(* Logix 5000 project; controller DispersionPlc vendor 1 type 14 code 108 rev 34.11; software revision 34.01; part 15 of 22 *)
(* tags used below, declared in another part *)
   _JISdebug : DINT;
   _Placeholder : DINT;
   AFI : BOOL;
   Estop_Disp : ALIAS FOR Local:3:I.Data.1;
   FQIC_4302_11_CurrentTrasferredLb : DINT;
   FQIC_4302_11_Reset : BOOL;
   FQIC_4302_11_TransferSetpoint : DINT;
   FQIC_4302_11_TransferStopValueLb : DINT;
   GenPurp : AStd_GeneralPurp;
   HS_S51_1 : AStd_DiscreteInput;
   HS_S51_1_AOI : AStd_DI_AOI;
   HS_S51_1_IRaw : BOOL;
   HS_S51_2 : AStd_DiscreteInput;
   HS_S51_2_AOI : AStd_DI_AOI;
   LAH_4302_11 : BOOL;   // Truck Loading Level Alarm High Probe
   LS_S51_1 : AStd_DiscreteInput;
   LS_S51_1_AOI : AStd_DI_AOI;
   LS_S51_1_IRaw : BOOL;
   LVL_W2_High : ALIAS FOR Local:1:I.Data[1].22;
   LVL_W4_High : ALIAS FOR Local:1:I.Data[1].23;
   PackTransferCompletePB : BOOL;
   RG_T51 : REAL;
   S4352_Phase_Circulation : AStd_PLI;
   S4352_Phase_Packaging_Transfer : AStd_PLI;
   S4352_Phase_Packaging_Transfer_AOI : AStd_PLI_AOI;
   S4352_Phase_TT_Transfer : AStd_PLI;
   S4352_Phase_TT_Transfer_AOI : AStd_PLI_AOI;
   S52TotalizerBypassPB : BOOL;
   SPARE_I_1_4_6 : ALIAS FOR Local:1:I.Data[4].6;
   SPARE_O_1_1_2 : ALIAS FOR Local:1:O.Data[1].2;
   SPARE_O_1_1_3 : ALIAS FOR Local:1:O.Data[1].3;
   SV_S52_2 : AStd_VlvOC;
   T4302_Phase_S52_Transfer : AStd_PLI;
   TIT_S51_1 : AStd_AnalogInput;
   TIT_S51_1_AOI : AStd_AI_AOI;
   TIT_S51_1_Raw : DINT;
   TIT_S51_2 : AStd_AnalogInput;
   TIT_S51_3 : AStd_AnalogInput;
   XV_4302_12 : AStd_VlvOC;
   XV_4302_13 : AStd_VlvOC;
   XV_S51_1 : AStd_VlvOC;
   XV_S51_1_AOI : AStd_VlvOC_AOI;
   XV_S51_1_IOpn : BOOL;
   XV_S51_1_OCls : BOOL;
   XV_S51_2 : AStd_VlvOC;
   XV_S51_2_AOI : AStd_VlvOC_AOI;
   XV_S51_2_ClsI : BOOL;
   XV_S51_2_IOpn : BOOL;
   XV_S51_2_OCls : BOOL;
   XV_S51_2CloseC : BOOL;
   XV_S51_2OpenC : BOOL;
   XV_S51_3 : AStd_VlvOC;
   XV_S51_3_AOI : AStd_VlvOC_AOI;
   XV_S51_3_IOpn : BOOL;
   XV_S51_3_OCls : BOOL;
   XV_S51_3CloseC : BOOL;
   XV_S51_3OpenC : BOOL;
   XV_S51_4 : AStd_VlvOC;
   XV_S51_4_AOI : AStd_VlvOC_AOI;
   XV_S51_4_IOpn : BOOL;
   XV_S51_4_OCls : BOOL;
   XV_S52_1 : AStd_VlvOC;
   XV_S52_2 : AStd_VlvOC;
(* Unit_S4352, continued *)

ROUTINE Phase_Packaging_Transfer   (* ladder *)
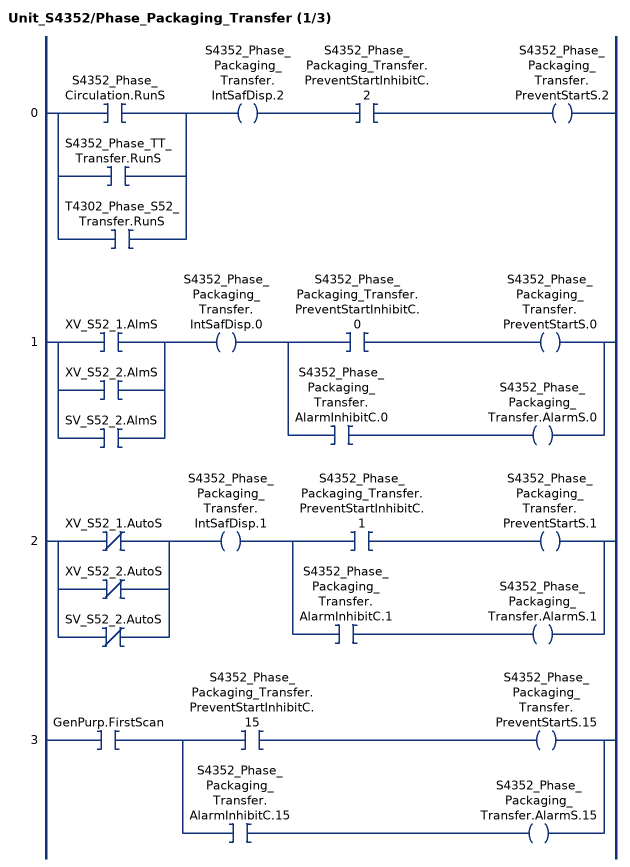
   0: [XIC(S4352_Phase_Circulation.RunS) ,XIC(S4352_Phase_TT_Transfer.RunS) ,XIC(T4302_Phase_S52_Transfer.RunS) ]OTE(S4352_Phase_Packaging_Transfer.IntSafDisp.2)XIC(S4352_Phase_Packaging_Transfer.PreventStartInhibitC.2)OTE(S4352_Phase_Packaging_Transfer.PreventStartS.2);
   1: [XIC(XV_S52_1.AlmS) ,XIC(XV_S52_2.AlmS) ,XIC(SV_S52_2.AlmS) ]OTE(S4352_Phase_Packaging_Transfer.IntSafDisp.0)[XIC(S4352_Phase_Packaging_Transfer.PreventStartInhibitC.0) OTE(S4352_Phase_Packaging_Transfer.PreventStartS.0) ,XIC(S4352_Phase_Packaging_Transfer.AlarmInhibitC.0) OTE(S4352_Phase_Packaging_Transfer.AlarmS.0) ];
   2: [XIO(XV_S52_1.AutoS) ,XIO(XV_S52_2.AutoS) ,XIO(SV_S52_2.AutoS) ]OTE(S4352_Phase_Packaging_Transfer.IntSafDisp.1)[XIC(S4352_Phase_Packaging_Transfer.PreventStartInhibitC.1) OTE(S4352_Phase_Packaging_Transfer.PreventStartS.1) ,XIC(S4352_Phase_Packaging_Transfer.AlarmInhibitC.1) OTE(S4352_Phase_Packaging_Transfer.AlarmS.1) ];
   3: XIC(GenPurp.FirstScan)[XIC(S4352_Phase_Packaging_Transfer.PreventStartInhibitC.15) OTE(S4352_Phase_Packaging_Transfer.PreventStartS.15) ,XIC(S4352_Phase_Packaging_Transfer.AlarmInhibitC.15) OTE(S4352_Phase_Packaging_Transfer.AlarmS.15) ];
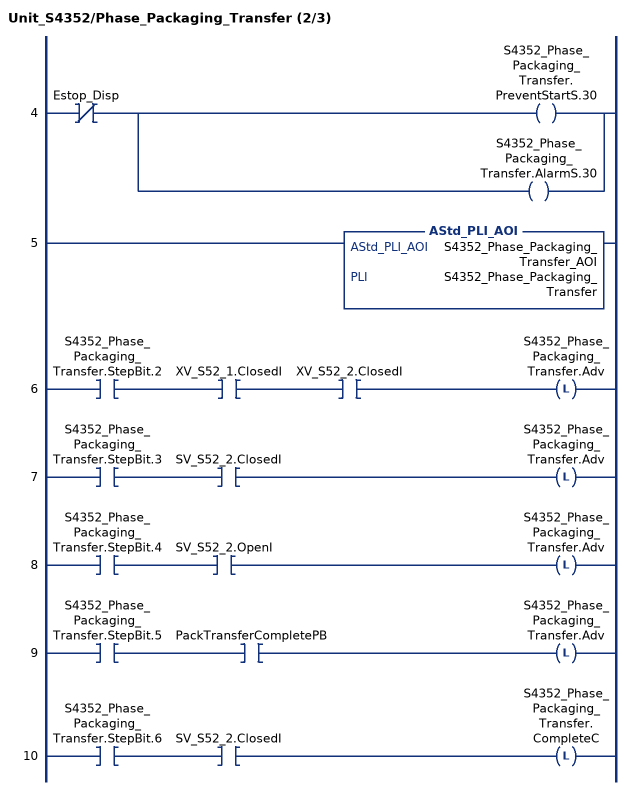
   4: XIO(Estop_Disp)[OTE(S4352_Phase_Packaging_Transfer.PreventStartS.30) ,OTE(S4352_Phase_Packaging_Transfer.AlarmS.30) ];
   5: AStd_PLI_AOI(S4352_Phase_Packaging_Transfer_AOI,S4352_Phase_Packaging_Transfer);
   6: XIC(S4352_Phase_Packaging_Transfer.StepBit.2)XIC(XV_S52_1.ClosedI)XIC(XV_S52_2.ClosedI)OTL(S4352_Phase_Packaging_Transfer.Adv);
   7: XIC(S4352_Phase_Packaging_Transfer.StepBit.3)XIC(SV_S52_2.ClosedI)OTL(S4352_Phase_Packaging_Transfer.Adv);
   8: XIC(S4352_Phase_Packaging_Transfer.StepBit.4)XIC(SV_S52_2.OpenI)OTL(S4352_Phase_Packaging_Transfer.Adv);
   9: XIC(S4352_Phase_Packaging_Transfer.StepBit.5)XIC(PackTransferCompletePB)OTL(S4352_Phase_Packaging_Transfer.Adv);
   10: XIC(S4352_Phase_Packaging_Transfer.StepBit.6)XIC(SV_S52_2.ClosedI)OTL(S4352_Phase_Packaging_Transfer.CompleteC);
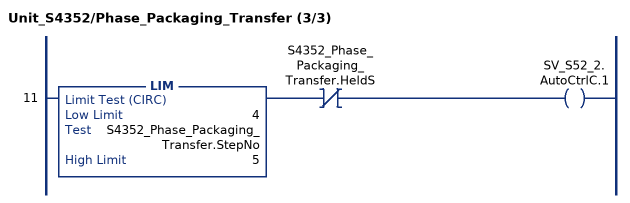
   11: LIM(4,S4352_Phase_Packaging_Transfer.StepNo,5)XIO(S4352_Phase_Packaging_Transfer.HeldS)OTE(SV_S52_2.AutoCtrlC.1);
END_ROUTINE

ROUTINE Phase_TT_Transfer   (* ladder *)
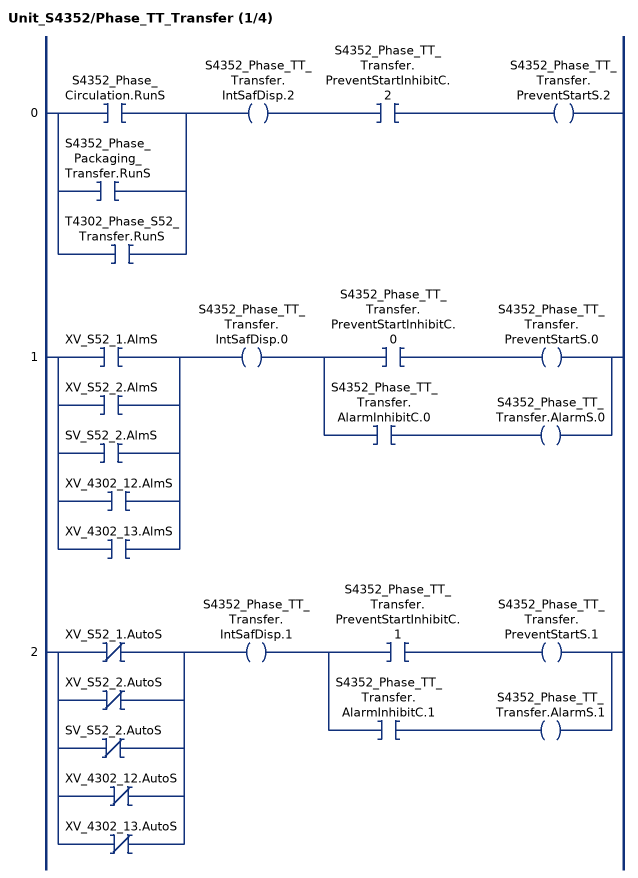
   0: [XIC(S4352_Phase_Circulation.RunS) ,XIC(S4352_Phase_Packaging_Transfer.RunS) ,XIC(T4302_Phase_S52_Transfer.RunS) ]OTE(S4352_Phase_TT_Transfer.IntSafDisp.2)XIC(S4352_Phase_TT_Transfer.PreventStartInhibitC.2)OTE(S4352_Phase_TT_Transfer.PreventStartS.2);
   1: [XIC(XV_S52_1.AlmS) ,XIC(XV_S52_2.AlmS) ,XIC(SV_S52_2.AlmS) ,XIC(XV_4302_12.AlmS) ,XIC(XV_4302_13.AlmS) ]OTE(S4352_Phase_TT_Transfer.IntSafDisp.0)[XIC(S4352_Phase_TT_Transfer.PreventStartInhibitC.0) OTE(S4352_Phase_TT_Transfer.PreventStartS.0) ,XIC(S4352_Phase_TT_Transfer.AlarmInhibitC.0) OTE(S4352_Phase_TT_Transfer.AlarmS.0) ];
   2: [XIO(XV_S52_1.AutoS) ,XIO(XV_S52_2.AutoS) ,XIO(SV_S52_2.AutoS) ,XIO(XV_4302_12.AutoS) ,XIO(XV_4302_13.AutoS) ]OTE(S4352_Phase_TT_Transfer.IntSafDisp.1)[XIC(S4352_Phase_TT_Transfer.PreventStartInhibitC.1) OTE(S4352_Phase_TT_Transfer.PreventStartS.1) ,XIC(S4352_Phase_TT_Transfer.AlarmInhibitC.1) OTE(S4352_Phase_TT_Transfer.AlarmS.1) ];
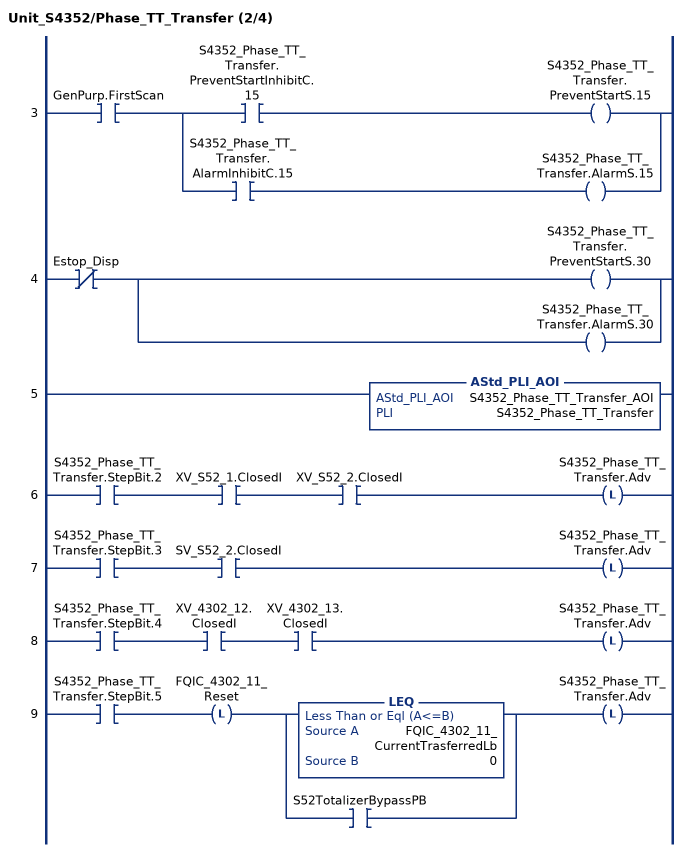
   3: XIC(GenPurp.FirstScan)[XIC(S4352_Phase_TT_Transfer.PreventStartInhibitC.15) OTE(S4352_Phase_TT_Transfer.PreventStartS.15) ,XIC(S4352_Phase_TT_Transfer.AlarmInhibitC.15) OTE(S4352_Phase_TT_Transfer.AlarmS.15) ];
   4: XIO(Estop_Disp)[OTE(S4352_Phase_TT_Transfer.PreventStartS.30) ,OTE(S4352_Phase_TT_Transfer.AlarmS.30) ];
   5: AStd_PLI_AOI(S4352_Phase_TT_Transfer_AOI,S4352_Phase_TT_Transfer);
   6: XIC(S4352_Phase_TT_Transfer.StepBit.2)XIC(XV_S52_1.ClosedI)XIC(XV_S52_2.ClosedI)OTL(S4352_Phase_TT_Transfer.Adv);
   7: XIC(S4352_Phase_TT_Transfer.StepBit.3)XIC(SV_S52_2.ClosedI)OTL(S4352_Phase_TT_Transfer.Adv);
   8: XIC(S4352_Phase_TT_Transfer.StepBit.4)XIC(XV_4302_12.ClosedI)XIC(XV_4302_13.ClosedI)OTL(S4352_Phase_TT_Transfer.Adv);
   9: XIC(S4352_Phase_TT_Transfer.StepBit.5)OTL(FQIC_4302_11_Reset)[LEQ(FQIC_4302_11_CurrentTrasferredLb,0) ,XIC(S52TotalizerBypassPB) ]OTL(S4352_Phase_TT_Transfer.Adv);
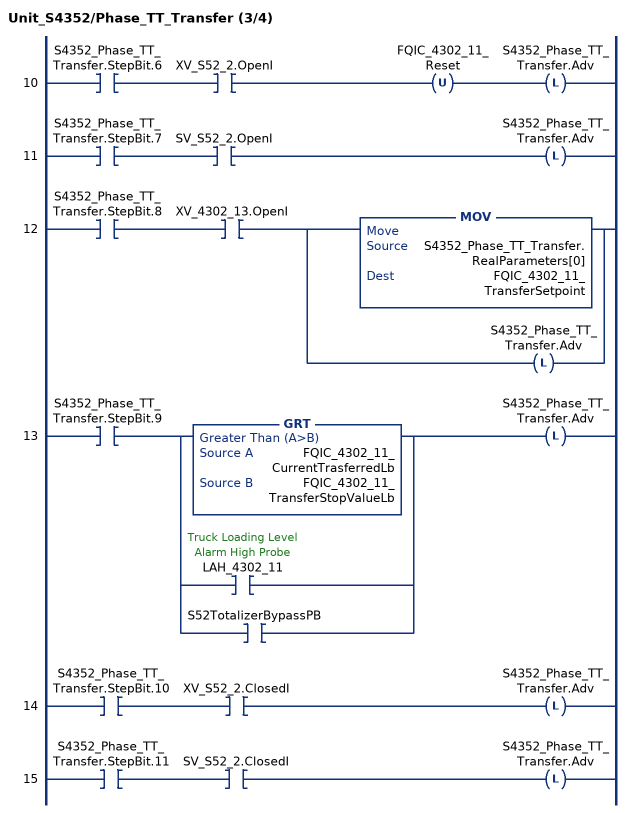
   10: XIC(S4352_Phase_TT_Transfer.StepBit.6)XIC(XV_S52_2.OpenI)OTU(FQIC_4302_11_Reset)OTL(S4352_Phase_TT_Transfer.Adv);
   11: XIC(S4352_Phase_TT_Transfer.StepBit.7)XIC(SV_S52_2.OpenI)OTL(S4352_Phase_TT_Transfer.Adv);
   12: XIC(S4352_Phase_TT_Transfer.StepBit.8)XIC(XV_4302_13.OpenI)[MOV(S4352_Phase_TT_Transfer.RealParameters[0],FQIC_4302_11_TransferSetpoint) ,OTL(S4352_Phase_TT_Transfer.Adv) ];
   13: XIC(S4352_Phase_TT_Transfer.StepBit.9)[GRT(FQIC_4302_11_CurrentTrasferredLb,FQIC_4302_11_TransferStopValueLb) ,XIC(LAH_4302_11) ,XIC(S52TotalizerBypassPB) ]OTL(S4352_Phase_TT_Transfer.Adv);
   14: XIC(S4352_Phase_TT_Transfer.StepBit.10)XIC(XV_S52_2.ClosedI)OTL(S4352_Phase_TT_Transfer.Adv);
   15: XIC(S4352_Phase_TT_Transfer.StepBit.11)XIC(SV_S52_2.ClosedI)OTL(S4352_Phase_TT_Transfer.Adv);
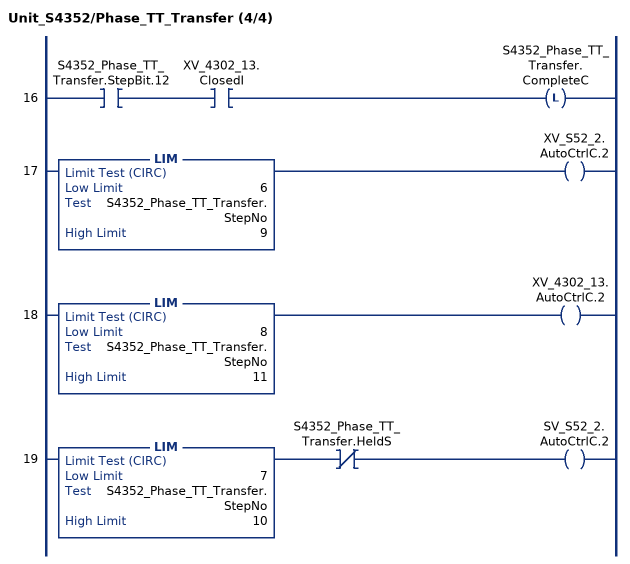
   16: XIC(S4352_Phase_TT_Transfer.StepBit.12)XIC(XV_4302_13.ClosedI)OTL(S4352_Phase_TT_Transfer.CompleteC);
   17: LIM(6,S4352_Phase_TT_Transfer.StepNo,9)OTE(XV_S52_2.AutoCtrlC.2);
   18: LIM(8,S4352_Phase_TT_Transfer.StepNo,11)OTE(XV_4302_13.AutoCtrlC.2);
   19: LIM(7,S4352_Phase_TT_Transfer.StepNo,10)XIO(S4352_Phase_TT_Transfer.HeldS)OTE(SV_S52_2.AutoCtrlC.2);
END_ROUTINE
END_PROGRAM

PROGRAM Unit_S51   (* main routine MainRoutine *)

ROUTINE Device_HS_S51_1   (* ladder *)
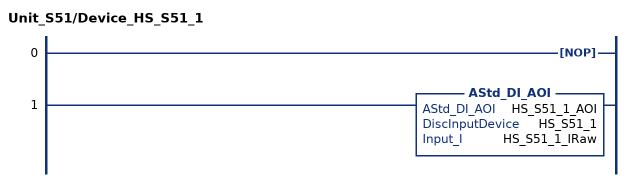
   0: NOP();
   1: AStd_DI_AOI(HS_S51_1_AOI,HS_S51_1,HS_S51_1_IRaw);
END_ROUTINE

ROUTINE Device_HS_S51_2   (* ladder *)
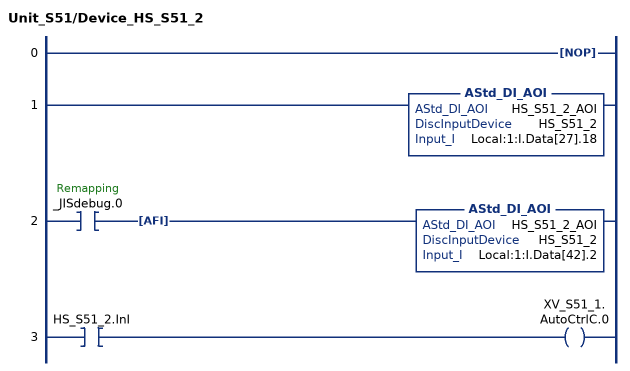
   0: NOP();
   1: AStd_DI_AOI(HS_S51_2_AOI,HS_S51_2,Local:1:I.Data[27].18);
   2: XIC(_JISdebug.0)AFI()AStd_DI_AOI(HS_S51_2_AOI,HS_S51_2,Local:1:I.Data[42].2);
   3: XIC(HS_S51_2.InI)OTE(XV_S51_1.AutoCtrlC.0);
END_ROUTINE

ROUTINE Device_LS_S51_1   (* ladder *)
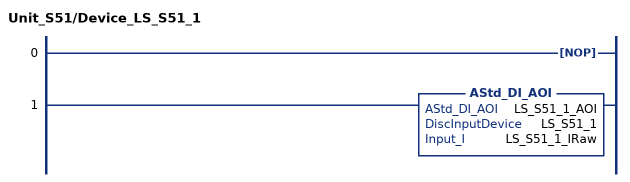
   0: NOP();
   1: AStd_DI_AOI(LS_S51_1_AOI,LS_S51_1,LS_S51_1_IRaw);
END_ROUTINE

ROUTINE Device_TIT_S51_1   (* ladder *)
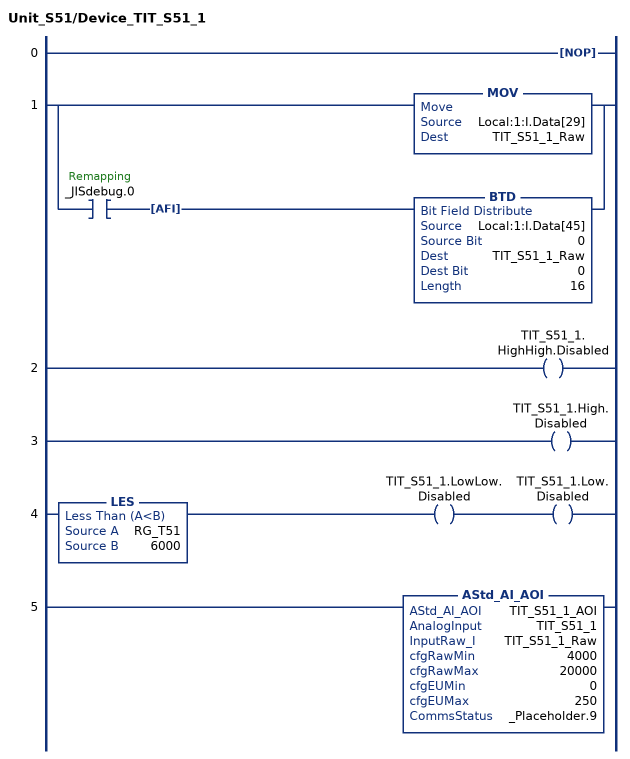
   0: NOP();
   1: [MOV(Local:1:I.Data[29],TIT_S51_1_Raw) ,XIC(_JISdebug.0) AFI() BTD(Local:1:I.Data[45],0,TIT_S51_1_Raw,0,16) ];
   2: OTE(TIT_S51_1.HighHigh.Disabled);
   3: OTE(TIT_S51_1.High.Disabled);
   4: LES(RG_T51,6000)OTE(TIT_S51_1.LowLow.Disabled)OTE(TIT_S51_1.Low.Disabled);
   5: AStd_AI_AOI(TIT_S51_1_AOI,TIT_S51_1,TIT_S51_1_Raw,4000,20000,0,250,_Placeholder.9);
END_ROUTINE

ROUTINE Device_XV_S51_1   (* ladder *)
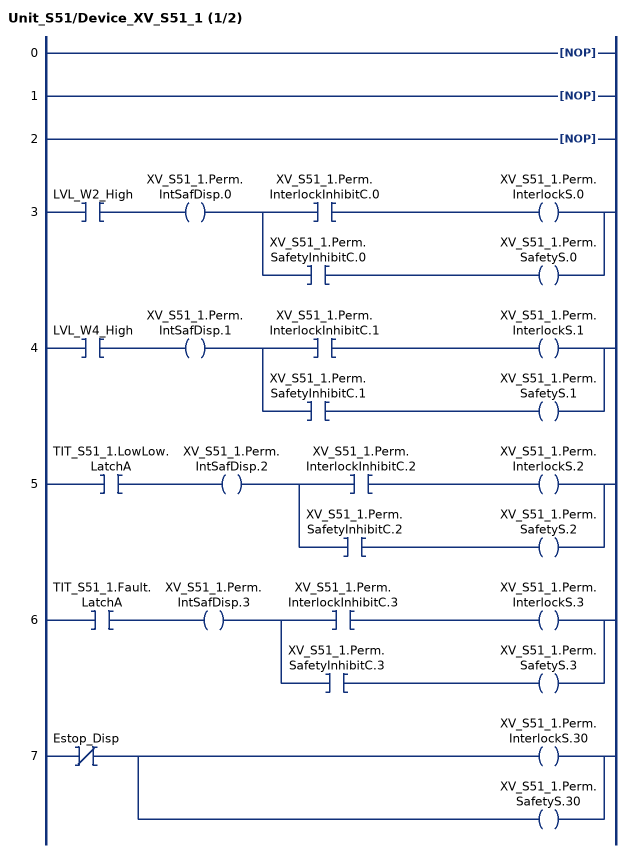
   0: NOP();
   1: NOP();
   2: NOP();
   3: XIC(LVL_W2_High)OTE(XV_S51_1.Perm.IntSafDisp.0)[XIC(XV_S51_1.Perm.InterlockInhibitC.0) OTE(XV_S51_1.Perm.InterlockS.0) ,XIC(XV_S51_1.Perm.SafetyInhibitC.0) OTE(XV_S51_1.Perm.SafetyS.0) ];
   4: XIC(LVL_W4_High)OTE(XV_S51_1.Perm.IntSafDisp.1)[XIC(XV_S51_1.Perm.InterlockInhibitC.1) OTE(XV_S51_1.Perm.InterlockS.1) ,XIC(XV_S51_1.Perm.SafetyInhibitC.1) OTE(XV_S51_1.Perm.SafetyS.1) ];
   5: XIC(TIT_S51_1.LowLow.LatchA)OTE(XV_S51_1.Perm.IntSafDisp.2)[XIC(XV_S51_1.Perm.InterlockInhibitC.2) OTE(XV_S51_1.Perm.InterlockS.2) ,XIC(XV_S51_1.Perm.SafetyInhibitC.2) OTE(XV_S51_1.Perm.SafetyS.2) ];
   6: XIC(TIT_S51_1.Fault.LatchA)OTE(XV_S51_1.Perm.IntSafDisp.3)[XIC(XV_S51_1.Perm.InterlockInhibitC.3) OTE(XV_S51_1.Perm.InterlockS.3) ,XIC(XV_S51_1.Perm.SafetyInhibitC.3) OTE(XV_S51_1.Perm.SafetyS.3) ];
   7: XIO(Estop_Disp)[OTE(XV_S51_1.Perm.InterlockS.30) ,OTE(XV_S51_1.Perm.SafetyS.30) ];
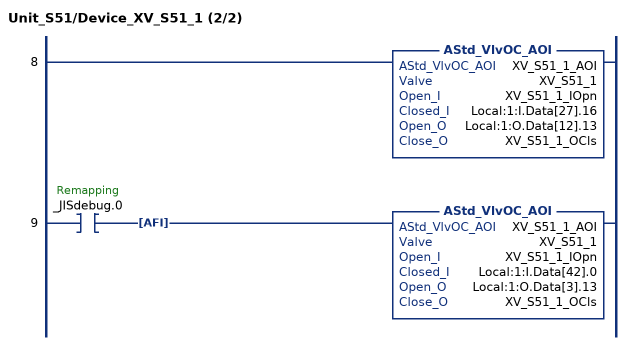
   8: AStd_VlvOC_AOI(XV_S51_1_AOI,XV_S51_1,XV_S51_1_IOpn,Local:1:I.Data[27].16,Local:1:O.Data[12].13,XV_S51_1_OCls);
   9: XIC(_JISdebug.0)AFI()AStd_VlvOC_AOI(XV_S51_1_AOI,XV_S51_1,XV_S51_1_IOpn,Local:1:I.Data[42].0,Local:1:O.Data[3].13,XV_S51_1_OCls);
END_ROUTINE

ROUTINE Device_XV_S51_2   (* ladder *)
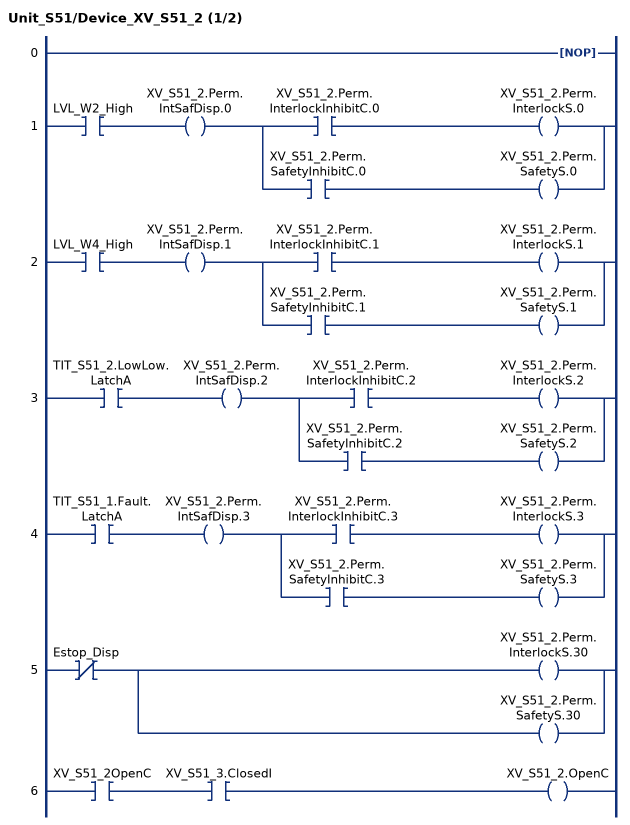
   0: NOP();
   1: XIC(LVL_W2_High)OTE(XV_S51_2.Perm.IntSafDisp.0)[XIC(XV_S51_2.Perm.InterlockInhibitC.0) OTE(XV_S51_2.Perm.InterlockS.0) ,XIC(XV_S51_2.Perm.SafetyInhibitC.0) OTE(XV_S51_2.Perm.SafetyS.0) ];
   2: XIC(LVL_W4_High)OTE(XV_S51_2.Perm.IntSafDisp.1)[XIC(XV_S51_2.Perm.InterlockInhibitC.1) OTE(XV_S51_2.Perm.InterlockS.1) ,XIC(XV_S51_2.Perm.SafetyInhibitC.1) OTE(XV_S51_2.Perm.SafetyS.1) ];
   3: XIC(TIT_S51_2.LowLow.LatchA)OTE(XV_S51_2.Perm.IntSafDisp.2)[XIC(XV_S51_2.Perm.InterlockInhibitC.2) OTE(XV_S51_2.Perm.InterlockS.2) ,XIC(XV_S51_2.Perm.SafetyInhibitC.2) OTE(XV_S51_2.Perm.SafetyS.2) ];
   4: XIC(TIT_S51_1.Fault.LatchA)OTE(XV_S51_2.Perm.IntSafDisp.3)[XIC(XV_S51_2.Perm.InterlockInhibitC.3) OTE(XV_S51_2.Perm.InterlockS.3) ,XIC(XV_S51_2.Perm.SafetyInhibitC.3) OTE(XV_S51_2.Perm.SafetyS.3) ];
   5: XIO(Estop_Disp)[OTE(XV_S51_2.Perm.InterlockS.30) ,OTE(XV_S51_2.Perm.SafetyS.30) ];
   6: XIC(XV_S51_2OpenC)XIC(XV_S51_3.ClosedI)OTE(XV_S51_2.OpenC);
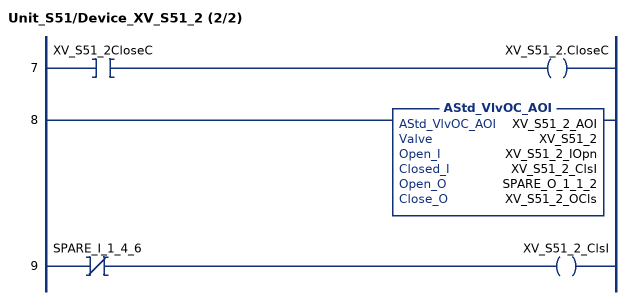
   7: XIC(XV_S51_2CloseC)OTE(XV_S51_2.CloseC);
   8: AStd_VlvOC_AOI(XV_S51_2_AOI,XV_S51_2,XV_S51_2_IOpn,XV_S51_2_ClsI,SPARE_O_1_1_2,XV_S51_2_OCls);
   9: XIO(SPARE_I_1_4_6)OTE(XV_S51_2_ClsI);
END_ROUTINE

ROUTINE Device_XV_S51_3   (* ladder *)
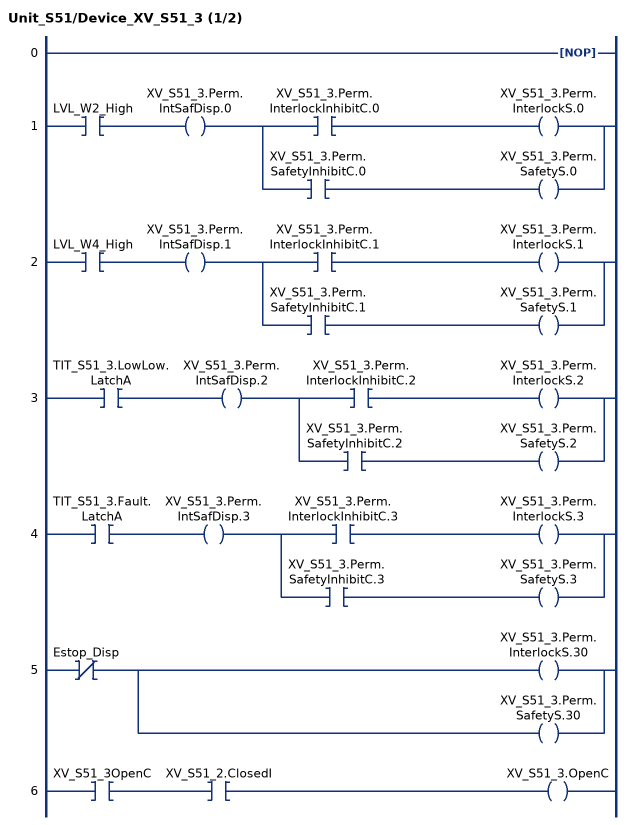
   0: NOP();
   1: XIC(LVL_W2_High)OTE(XV_S51_3.Perm.IntSafDisp.0)[XIC(XV_S51_3.Perm.InterlockInhibitC.0) OTE(XV_S51_3.Perm.InterlockS.0) ,XIC(XV_S51_3.Perm.SafetyInhibitC.0) OTE(XV_S51_3.Perm.SafetyS.0) ];
   2: XIC(LVL_W4_High)OTE(XV_S51_3.Perm.IntSafDisp.1)[XIC(XV_S51_3.Perm.InterlockInhibitC.1) OTE(XV_S51_3.Perm.InterlockS.1) ,XIC(XV_S51_3.Perm.SafetyInhibitC.1) OTE(XV_S51_3.Perm.SafetyS.1) ];
   3: XIC(TIT_S51_3.LowLow.LatchA)OTE(XV_S51_3.Perm.IntSafDisp.2)[XIC(XV_S51_3.Perm.InterlockInhibitC.2) OTE(XV_S51_3.Perm.InterlockS.2) ,XIC(XV_S51_3.Perm.SafetyInhibitC.2) OTE(XV_S51_3.Perm.SafetyS.2) ];
   4: XIC(TIT_S51_3.Fault.LatchA)OTE(XV_S51_3.Perm.IntSafDisp.3)[XIC(XV_S51_3.Perm.InterlockInhibitC.3) OTE(XV_S51_3.Perm.InterlockS.3) ,XIC(XV_S51_3.Perm.SafetyInhibitC.3) OTE(XV_S51_3.Perm.SafetyS.3) ];
   5: XIO(Estop_Disp)[OTE(XV_S51_3.Perm.InterlockS.30) ,OTE(XV_S51_3.Perm.SafetyS.30) ];
   6: XIC(XV_S51_3OpenC)XIC(XV_S51_2.ClosedI)OTE(XV_S51_3.OpenC);
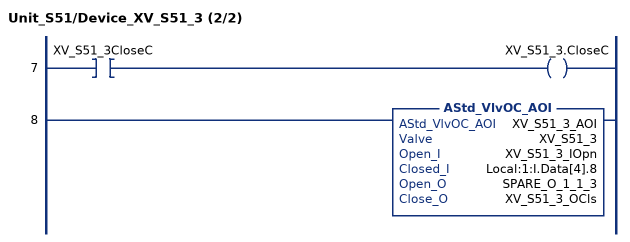
   7: XIC(XV_S51_3CloseC)OTE(XV_S51_3.CloseC);
   8: AStd_VlvOC_AOI(XV_S51_3_AOI,XV_S51_3,XV_S51_3_IOpn,Local:1:I.Data[4].8,SPARE_O_1_1_3,XV_S51_3_OCls);
END_ROUTINE

ROUTINE Device_XV_S51_4   (* ladder *)
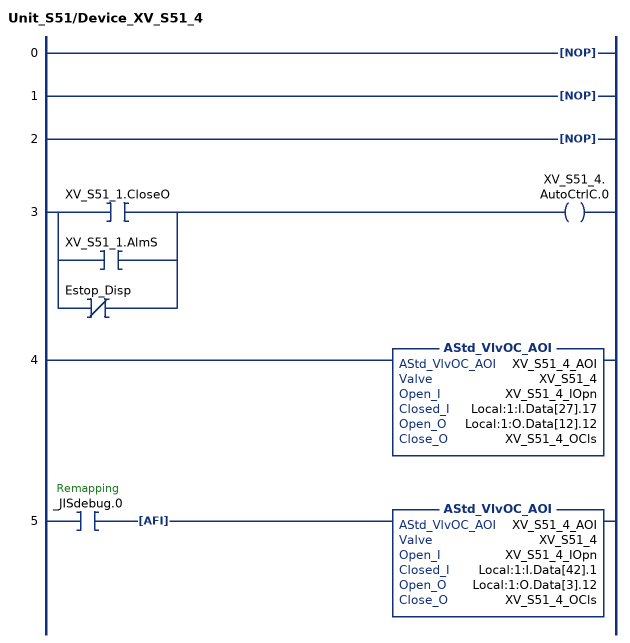
   0: NOP();
   1: NOP();
   2: NOP();
   3: [XIC(XV_S51_1.CloseO) ,XIC(XV_S51_1.AlmS) ,XIO(Estop_Disp) ]OTE(XV_S51_4.AutoCtrlC.0);
   4: AStd_VlvOC_AOI(XV_S51_4_AOI,XV_S51_4,XV_S51_4_IOpn,Local:1:I.Data[27].17,Local:1:O.Data[12].12,XV_S51_4_OCls);
   5: XIC(_JISdebug.0)AFI()AStd_VlvOC_AOI(XV_S51_4_AOI,XV_S51_4,XV_S51_4_IOpn,Local:1:I.Data[42].1,Local:1:O.Data[3].12,XV_S51_4_OCls);
END_ROUTINE
